PROGRAM MAIN

VAR
END_VAR

END_PROGRAM

(* stored: Version 1.1.0.1, ProductVersion 3.1.4024.12
   POU MAIN: Id {01a27337-1fc8-4097-a1a5-04fef61cf819}, SpecialFunc None *)
